// TIA Portal V20 export
// export: Created 2025-09-12T17:58:00.0000000Z, ExportSetting WithDefaults
FUNCTION_BLOCK "FB200_EM_Cooling"   // FB, SCL
TITLE = EM-200: Cooling Control
AUTHOR : Dallas Levine
VERSION : 0.1
// This block contains all logic for the Cooling Equipment Module (EM-200).
// stored: AutoNumber true, IsRetain false
   VAR_INPUT
      Enable : Bool;   // Enables the block's execution.
   END_VAR
   VAR
      UDT : "UDT200_EM_Cooling";   // The data interface for the Cooling Equipment Module.
   END_VAR
BEGIN
   REGION Placeholder for SCL Code 

   END_REGION
END_FUNCTION_BLOCK
